Staubli VAL3: parseStackInfo.pgx

program parseStackInfo(string stackInfo_, string& library_[], string& program_[], num& line_[], string& code_[])
  local bool error
  local string dummy
begin
    //
  //\var error
  //\var dummy
  //\param stackInfo_
  //\param library_
  //\param program_
  //\param line_
  //\param code_
  //
if len(stackInfo_)>0
    library_=left(stackInfo_,find(stackInfo_,":"))
    stackInfo_=right(stackInfo_,len(stackInfo_)-find(stackInfo_,":")-1)
    program_=left(stackInfo_,find(stackInfo_,")")+1)
    stackInfo_=right(stackInfo_,len(stackInfo_)-find(stackInfo_,")")-1)
    stackInfo_=right(stackInfo_,len(stackInfo_)-find(stackInfo_,"ne")-3)
    dummy=stackInfo_
    dummy=toNum(dummy,line_,error)
    stackInfo_=right(stackInfo_,len(stackInfo_)-find(stackInfo_,":")-1)
    code_=stackInfo_
  endIf
end
